{attribute 'linkalways'} 
{attribute 'no_explicit_call' := 'This FB is a CLASS and must be accessed using methods or properties'}
{attribute 'enable_dynamic_creation'}
FUNCTION_BLOCK JsonDeserializerNullObjectForwardEnumerator EXTENDS Disposable IMPLEMENTS I_DeserializerObjectForwardEnumerator, I_EventHandler
VAR
	parent : I_JsonDeserializer;
	nullNode : I_Deserializer;
	invalid : BOOL := FALSE; 
END_VAR

PROPERTY PUBLIC Current : I_Deserializer
GET
Current := nullNode;
END_GET
END_PROPERTY

METHOD FB_exit : BOOL
VAR_INPUT
	bInCopyCode : BOOL; // if TRUE, the exit method is called for exiting an instance that is copied afterwards (online change).
END_VAR
IF bInCopyCode THEN
	RETURN;
END_IF

IF parent = 0 THEN
	RETURN;
END_IF

parent.OffEvent('OnChanged',THIS^);
parent.OffEvent('OnDisposed',THIS^);
END_METHOD

METHOD FB_init : BOOL
VAR_INPUT
	bInitRetains : BOOL; // if TRUE, the retain variables are initialized (warm start / cold start)
	bInCopyCode : BOOL;  // if TRUE, the instance afterwards gets moved into the copy code (online change)
	ParentJsonDeserializer : I_JsonDeserializer;
	ParentNullDeserializer : I_Deserializer;
END_VAR
parent := ParentJsonDeserializer;
nullNode := ParentNullDeserializer;

parent.OnEvent('OnChanged',THIS^);
parent.OnEvent('OnDisposed',THIS^);
END_METHOD

METHOD PUBLIC HandleEvent
VAR_INPUT
	Event : I_Event;
END_VAR
VAR
	changedEvent : I_JsonDeserializerChangedEvent;
	disposedEvent : I_JsonDeserializerDisposedEvent;
END_VAR
IF __QUERYINTERFACE(Event, changedEvent) THEN
	invalid := TRUE;
ELSIF __QUERYINTERFACE(Event, disposedEvent) THEN
	parent := 0;
END_IF
END_METHOD

PROPERTY PUBLIC IsValid : BOOL
GET // PUBLIC
IsValid := (NOT invalid AND parent <> 0);
END_GET
END_PROPERTY

PROPERTY Key : T_MAXSTRING
GET
END_GET
END_PROPERTY

METHOD PUBLIC MoveNext : BOOL
MoveNext := FALSE;
END_METHOD

END_FUNCTION_BLOCK

(* stored: Version 1.1.0.1, ProductVersion 3.1.4024.12
   POU JsonDeserializerNullObjectForwardEnumerator: Id {440a46ff-f73d-4d01-9040-a9c98f96408a}, SpecialFunc None
   Folder Constructor: Id {83bd1184-d4f9-45f8-8f71-123c780cd078}
   Folder Destructor: Id {7503838f-4a7b-4e61-9d11-e9f44aab5d26}
   Property Current: Id {820971fd-bfd9-4a6f-b18b-b0336a053862}
   Get Get: Id {c7b7e92a-646b-4cf6-928d-a45ffb60cfb8}
   Method FB_exit: Id {77a71383-53ec-477e-8933-e4482a2cb87d}
   Method FB_init: Id {c35f5e0e-5c93-4301-984d-9c4784ce7cb8}
   Method HandleEvent: Id {edf032b9-7fd0-4a47-beeb-599ec2bf3cc5}
   Property IsValid: Id {8092d6fd-dac2-4d24-8c5c-a33aabe14a99}
   Get Get: Id {8316cb57-1a90-4072-a384-f0014b61dac7}
   Property Key: Id {d4c1d814-9a91-4d62-9f38-302eaa5eedcb}
   Get Get: Id {20381df7-b3ca-4183-a77b-640a764100e6}
   Method MoveNext: Id {bd9acc61-d4a4-49b4-8b96-5c83d726b708} *)
